// TIA Portal V19 export
TYPE "EFC_CONTROL_WORD"
   STRUCT
      FreeWheelingStop : Bool := false;
      TorqueControl : Bool := false;
      Reserved2 : Bool := false;
      Reserved3 : Bool := false;
      Reserved4 : Bool := false;
      Reserved5 : Bool := false;
      Reserved6 : Bool := false;
      Reserved7 : Bool := false;
      Run : Bool := false;
      Jog : Bool := false;
      Reverse : Bool := false;
      StopParameter : Bool := false;
      EStop : Bool := false;
      ErrorReset : Bool := false;
      StopAccDec : Bool := false;
      ControlWord : Bool := false;
   END_STRUCT;
END_TYPE
